FUNCTION_BLOCK FB_YesNo
VAR_INPUT
	bYes			: BOOL;
	bNo				: BOOL;
END_VAR
VAR_OUTPUT
	bAnswer			: BOOL;
	bGotAnswer		: BOOL;
END_VAR
VAR
	fTrig			: F_Trig;
	rTrig			: R_Trig;
END_VAR

rTrig(CLK := bYes);
fTrig(CLK := bNo);

IF (rTrig.Q OR fTrig.Q) THEN
	bGotAnswer := TRUE;
END_IF
IF bYes THEN
	bAnswer := TRUE;
END_IF

{attribute 'TcRpcEnable'}
METHOD Reset
bAnswer		:= FALSE;
bGotAnswer 	:= FALSE;
END_METHOD

END_FUNCTION_BLOCK

(* stored: Version 1.1.0.1, ProductVersion 3.1.4024.11
   POU FB_YesNo: Id {929bb7e6-d658-465b-94c7-36f425484edf}, SpecialFunc None
   Method Reset: Id {c77281e2-163c-4bf8-bbbb-fd08b0adff3d} *)
